// TIA Portal project "PLC-Lab-Edit-ProjectTemplate-1200-G2" (V20)

(* hardware
DEVICE "S7-1200 G2-Station_1"  S7-1200 G2 Station
   slot 0: "Baugruppenträger_0"  S71200G2 Rack  Rack  V1.0
   slot 1: "G2_PLC_1"  CPU 1212C DC/DC/DC  6ES7 212-1AG50-0XB0  V1.0
   slot 2: "SM 1221 DI16 x DC24V_1"  SM 1221 DI16 x 24VDC  6ES7 221-1BH50-0XB0  V1.0
*)

// ===== PLC "G2_PLC_1"  CPU 1212C DC/DC/DC =====

FUNCTION "MHJ-PLC-Lab-Function-S71200-G2" : Void   // FC1, SCL
{ S7_Optimized_Access := 'TRUE' }
VERSION : 0.1
   VAR_INPUT
      MinDiByte : Int;
      MaxDiByte : Int;
   END_VAR
   VAR_TEMP
      Value : Byte;
      ForCounter : Int;
      MaxDiByteTemp : Int;
      MinDiByteTemp : Int;
   END_VAR
   VAR CONSTANT
      Value_01_DW : DWord := 16#1223_5486;
      Value_02_DW : DWord := 16#A6C9_D1F5;
   END_VAR
BEGIN

   #Value:=PEEK(area := 16#82,
        dbNumber := 0,
        byteOffset := 511);
   #Value := #Value + 1;

   POKE(area := 16#82,
        dbNumber := 0,
        byteOffset := 511,
        value := #Value);

   POKE(area := 16#82,
        dbNumber := 0,
        byteOffset := 1016,
        value := #Value_01_DW);
   POKE(area := 16#82,
        dbNumber := 0,
        byteOffset := 1020,
        value := #Value_02_DW);

   #MaxDiByteTemp := 462;
   IF #MaxDiByte < 463 THEN
       #MaxDiByteTemp := #MaxDiByte;
   END_IF;

   #MinDiByteTemp := 0;
   IF #MaxDiByteTemp >= #MinDiByte & #MinDiByte >= 0 THEN
       #MinDiByteTemp := #MinDiByte;
   END_IF;

   FOR #ForCounter := #MinDiByteTemp TO #MaxDiByteTemp DO
       #Value := PEEK(area := 16#1,
                      dbNumber := 0,
                      byteOffset := #ForCounter);
       POKE(area := 16#81,
            dbNumber := 0,
            byteOffset := #ForCounter,
            value := #Value);
   END_FOR;

   #Value := PEEK(area := 16#1,
                  dbNumber := 0,
                  byteOffset := 512);
   POKE(area := 16#82,
        dbNumber := 0,
        byteOffset := 512,
        value := #Value);
END_FUNCTION

FUNCTION "MHJ-PLC-Lab-Function-S71200-G2-NextInputArea" : Void   // FC2, SCL
{ S7_Optimized_Access := 'TRUE' }
VERSION : 0.1
   VAR_INPUT
      MinDiByte : Int;
      MaxDiByte : Int;
   END_VAR
   VAR_TEMP
      Value : Byte;
      ForCounter : Int;
      MaxDiByteTemp : Int;
      MinDiByteTemp : Int;
   END_VAR
BEGIN


   #MaxDiByteTemp := -1;
   IF #MaxDiByte < 463 THEN
       #MaxDiByteTemp := #MaxDiByte;
   END_IF;

   #MinDiByteTemp := -1;
   IF #MaxDiByteTemp >= #MinDiByte & #MinDiByte >= 0 THEN
       #MinDiByteTemp := #MinDiByte;
   END_IF;

   IF #MaxDiByteTemp >= 0 & #MinDiByte >= 0 THEN
       FOR #ForCounter := #MinDiByteTemp TO #MaxDiByteTemp DO
           #Value := PEEK(area := 16#1,
                          dbNumber := 0,
                          byteOffset := #ForCounter);
           POKE(area := 16#81,
                dbNumber := 0,
                byteOffset := #ForCounter,
                value := #Value);
       END_FOR;

   END_IF;
END_FUNCTION

ORGANIZATION_BLOCK "Main"   // OB1, FBD, ProgramCycle
TITLE = "Main Program Sweep (Cycle)"
{ S7_Optimized_Access := 'TRUE' }
VERSION : 0.1
   VAR_INPUT
      Initial_Call : Bool;   // Initial call of this OB
      Remanence : Bool;   // =True, if remanent data are available
   END_VAR
BEGIN

REGION Network 1
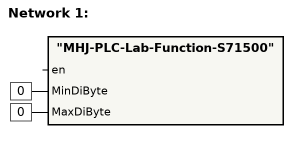
   "MHJ-PLC-Lab-Function-S71500"(MinDiByte := 0, MaxDiByte := 0);
END_REGION
END_ORGANIZATION_BLOCK